FUNCTION_BLOCK AUDI_UDINT_GT (* greater than *)
  (* Standard: 61131-3; Classification: standard comparison function; Description: Copyright (c) 2013 TU Wien ACIN\n \nThis program and the accompanying materials are made\navailable under the terms of the Eclipse Public License 2.0\nwhich is available at https://www.eclipse.org/legal/epl-2.0/\n\nSPDX-License-Identifier: EPL-2.0 *)
  (* Version 3.0, 2025-04-14, Patrick Aigner, changed package *)
  (* Version 1.0, 2013-03-13, Monika Wenger, TU Wien ACIN *)
  PACKAGE adapter::iec61131::comparison;
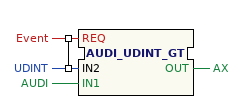
  EVENT_INPUT
    REQ WITH IN2; (* Service Request *)
  END_EVENT
  VAR_INPUT
    IN2 : UDINT; (* Input value 2 *)
  END_VAR
  SOCKETS
    IN1 : adapter::types::unidirectional::AUDI; (* Input value 1 *)
  END_SOCKETS
  PLUGS
    OUT : adapter::types::unidirectional::AX; (* value 1 > value2 = true *)
  END_PLUGS
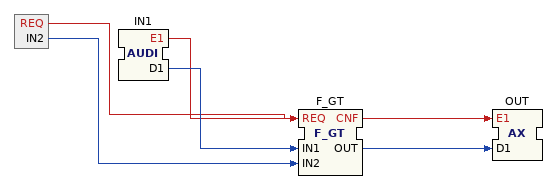
  FBS
    F_GT : iec61131::comparison::F_GT;
  END_FBS
  EVENT_CONNECTIONS
    F_GT.CNF TO OUT.E1;
    IN1.E1 TO F_GT.REQ;
    REQ TO F_GT.REQ;
  END_CONNECTIONS
  DATA_CONNECTIONS
    F_GT.OUT TO OUT.D1;
    IN1.D1 TO F_GT.IN1;
    IN2 TO F_GT.IN2;
  END_CONNECTIONS
END_FUNCTION_BLOCK
